# EPICS substitutions: ipimbLib/Db/bldFanout.substitutions
file bldFanout.db
{
  pattern { "" }
  { "" }
}
